Staubli VAL3: RobotStatus.pjx

Parameters version=s7.9.1 stackSize=5000 millimeterUnit=true
Data file=RobotStatus.dtx
Type name=JointSpace path=./JointSpace/JointSpace.pjx
Type name=CartesianSpace path=./CartesianSpace/CartesianSpace.pjx
